Universal Robots PolyScope program: prueba_visionsimple.urp

Program prueba_visionsimple (installation=default directory=/programs/usbdisk createdIn=5.12.5.1101767 lastSavedIn=5.12.5.1101767 robotSerialNumber=20215500624)
Calibrated DH parameters: a=[0.000186, -0.025908, -0.392311, -0.000071, 0.00009, 0]; d=[0.162736, -361.104072, 360.092318, 1.145413, 0.099738, 0.099626]; alpha=[1.57079, -0.001175, 0.009075, 1.569386, -1.569463, 0]; deltaTheta=[0, 1.509811, 4.749978, 0.023394, 0, -0.000001]
BeforeStart
  conexion := False
  datos_socket := [0,0,0,0]
  datos_posicion := datos_socket
  pos_base_camara := p[0,0,0,0,0,0]
  pos_pick := p[0,0,0,0,0,0]
Robot Program (runOnlyOnce=false)
  MoveJ speed 60 deg/s, acceleration 80 deg/s^2 (useActiveTCP=true) feature=Base
    Waypoint punto_ref: TCP in base x=111.932 y=-754.32 z=406.98 mm, rx=1.8017 ry=1.5729 rz=-0.3587 rad; joints [-71.902, -107.187, -82.163, -36.064, 91.458, 116.727] deg; TCP offset x=0 y=0 z=138.6 mm, rx=0 ry=0 rz=0 rad
  Folder Apertura socket
    Loop While (checkContinuously=false) expression=conexion≟ False
      conexion := socket_open("192.168.1.249",50000)
      Wait Sleep waitTime=0.01
  Folder Envío cadena socket
    str := "Listo"
    Script: socket_send_line(str)
  Call Lectura_de_datos_socket
  Folder Calcular pos_pick
    pos_pick := pose_trans(punto_ref,pos_base_camara)
  Folder Mover a pos_pick
    MoveJ speed 60 deg/s, acceleration 80 deg/s^2 (useActiveTCP=true) feature=Base
      Waypoint Punto_de_paso (Variable): variable(name=pos_pick)
SubProgram -> Lectura_de_datos_socket
SubProgram Lectura_de_datos_socket (keepSynchronizedWithDisk=false)
  Loop While (checkContinuously=false) expression=datos_socket[0]≠3
    datos_socket := socket_read_ascii_float(3)
    Wait Sleep waitTime=0.5
  Folder Asignación variables
    x := datos_socket[1]
    y := datos_socket[2]
    rz := datos_socket[3]
    'Convertir mm a m y deg a rad'
    pos_base_camara := p[x/1000,y/1000,0,0,0,d2r(rz)]
    datos_socket := [0,0,0,0]
